// TIA Portal V17 export
// export: Created 2024-09-02T12:50:06.6332122Z, ExportSetting WithDefaults, DisplayName Totally Integrated Automation Portal, DisplayVersion V17, DisplayName TIA Portal Openness, DisplayVersion V17, DisplayName TIA Portal Version Control Interface, DisplayVersion V17, DisplayName STEP 7 Professional, DisplayVersion V17, DisplayName STEP 7 Safety, DisplayVersion V17, DisplayName WinCC Professional, DisplayVersion V17
FUNCTION_BLOCK "GraFB2_FG01_Station_OP70"   // FB1282, GRAPH
VERSION : 0.1
// stored: AcknowledgeErrorsRequired false, AutoNumber false, GraphVersion 4.0, InitialValuesAcquisition true, IsIECCheckEnabled false, LanguageInNetworks LAD, LockOperatingMode false, PermanentILProcessingInMANMode true, SetENOAutomatically false, SkipSteps false, UDAEnableTagReadback false, WithAlarmHandling true
   // inherited from GRAPH_BASE
   VAR
      OFF_SQ_BASE : Bool;
   END_VAR
   VAR_INPUT
      OFF_SQ { ExternalWritable := 'False'} : Bool := false;
      INIT_SQ { ExternalWritable := 'False'} : Bool := false;
      ACK_EF { ExternalWritable := 'False'} : Bool := false;
      S_PREV { ExternalWritable := 'False'} : Bool := false;
      S_NEXT { ExternalWritable := 'False'} : Bool := false;
      SW_AUTO { ExternalWritable := 'False'} : Bool := false;
      SW_TAP { ExternalWritable := 'False'} : Bool := false;
      SW_TOP { ExternalWritable := 'False'} : Bool := false;
      SW_MAN { ExternalWritable := 'False'} : Bool := false;
      S_SEL { ExternalWritable := 'False'} : Int := 0;
      S_ON { ExternalWritable := 'False'} : Bool := false;
      S_OFF { ExternalWritable := 'False'} : Bool := false;
      T_PUSH { ExternalWritable := 'False'} : Bool := false;
   END_VAR
   VAR_OUTPUT
      S_NO { ExternalWritable := 'False'} : Int := 0;
      S_MORE { ExternalWritable := 'False'} : Bool := false;
      S_ACTIVE { ExternalWritable := 'False'} : Bool := false;
      ERR_FLT { ExternalWritable := 'False'} : Bool := false;
      AUTO_ON { ExternalWritable := 'False'} : Bool := false;
      TAP_ON { ExternalWritable := 'False'} : Bool := false;
      TOP_ON { ExternalWritable := 'False'} : Bool := false;
      MAN_ON { ExternalWritable := 'False'} : Bool := false;
   END_VAR
   VAR
      extBlock { S7_SetPoint := 'True'} : "LTLL_ManualGraphExt";
   END_VAR
BEGIN
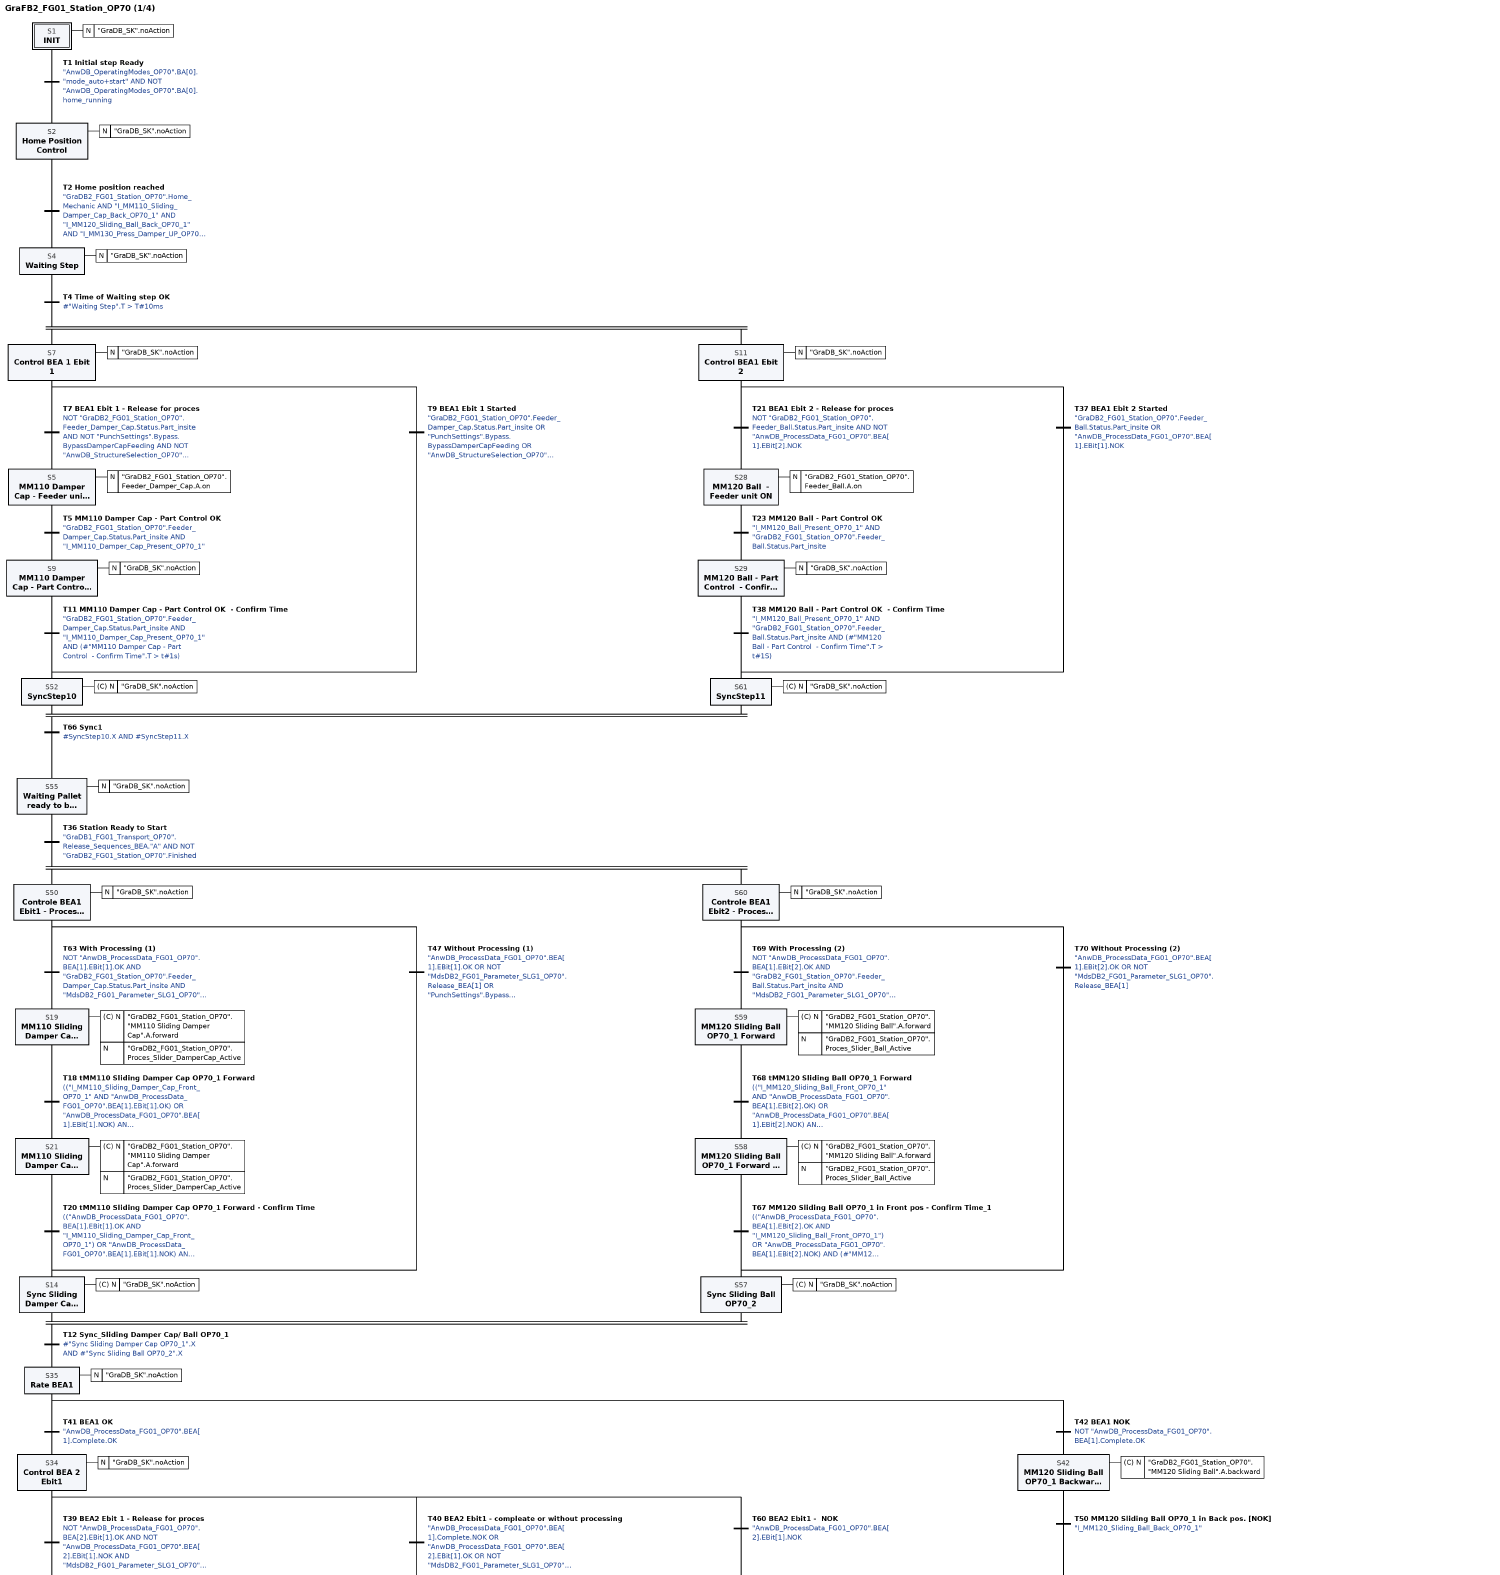
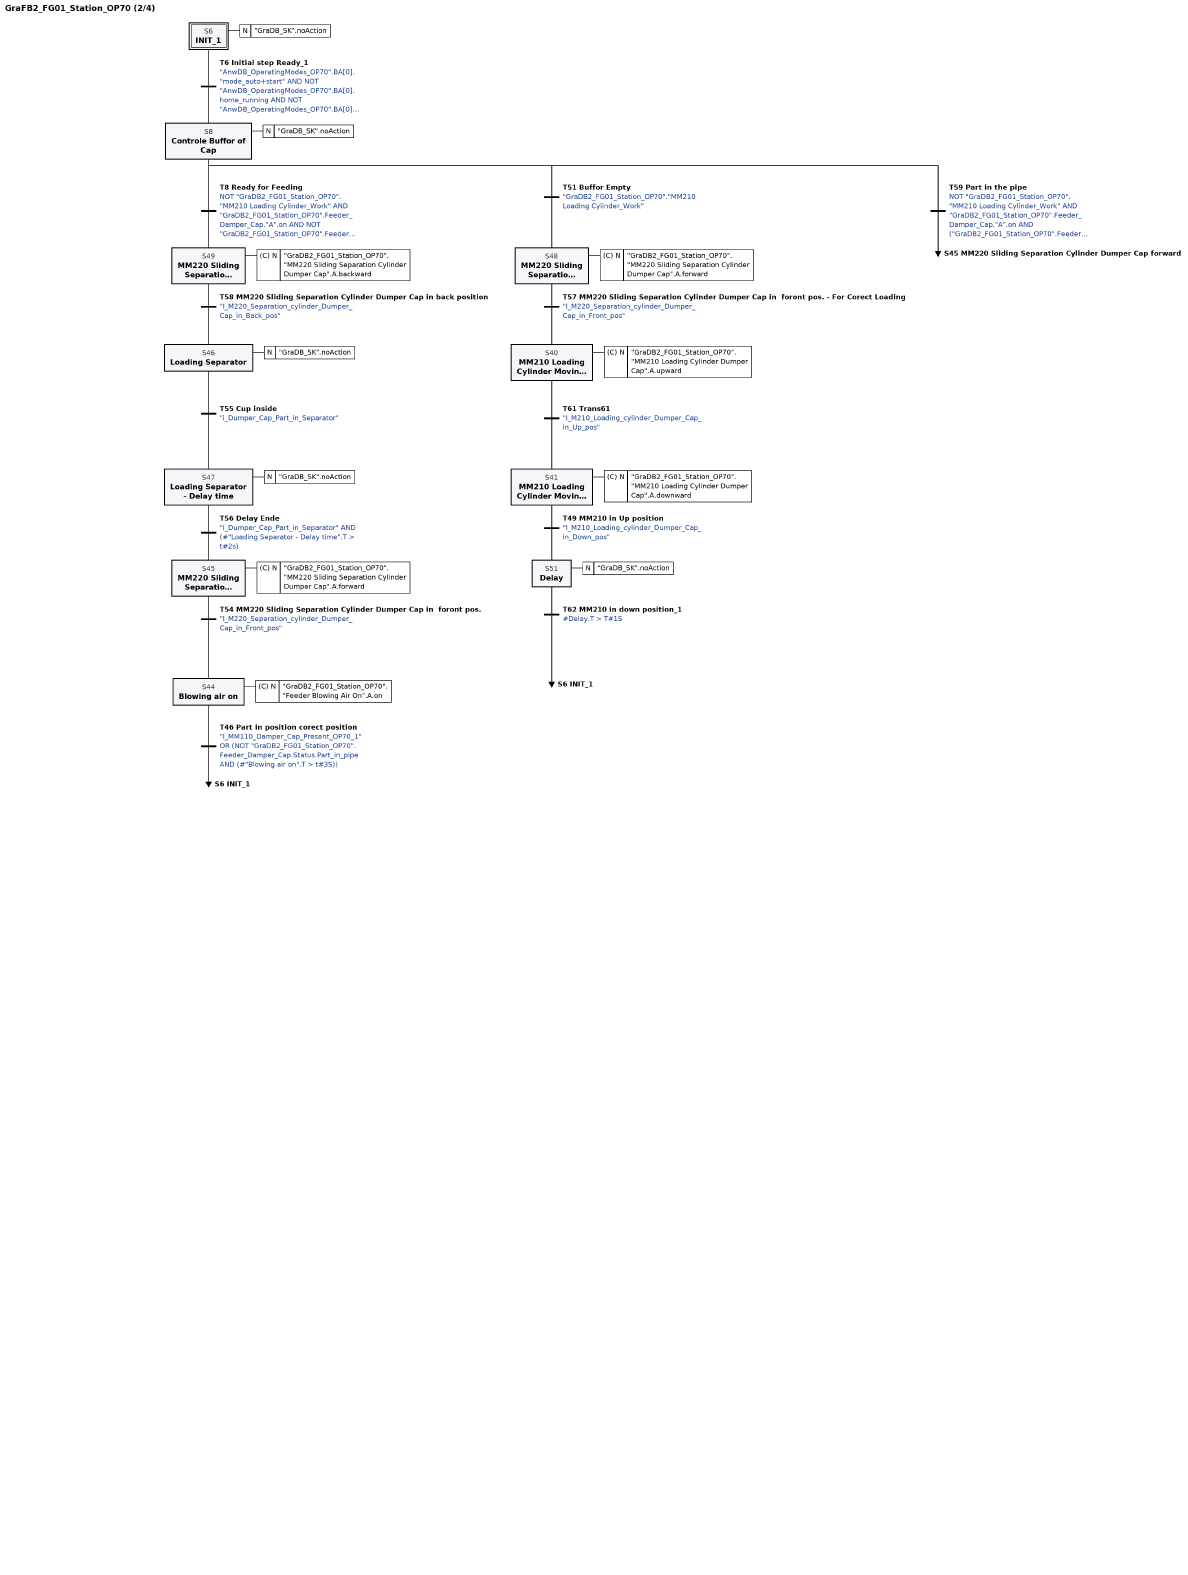
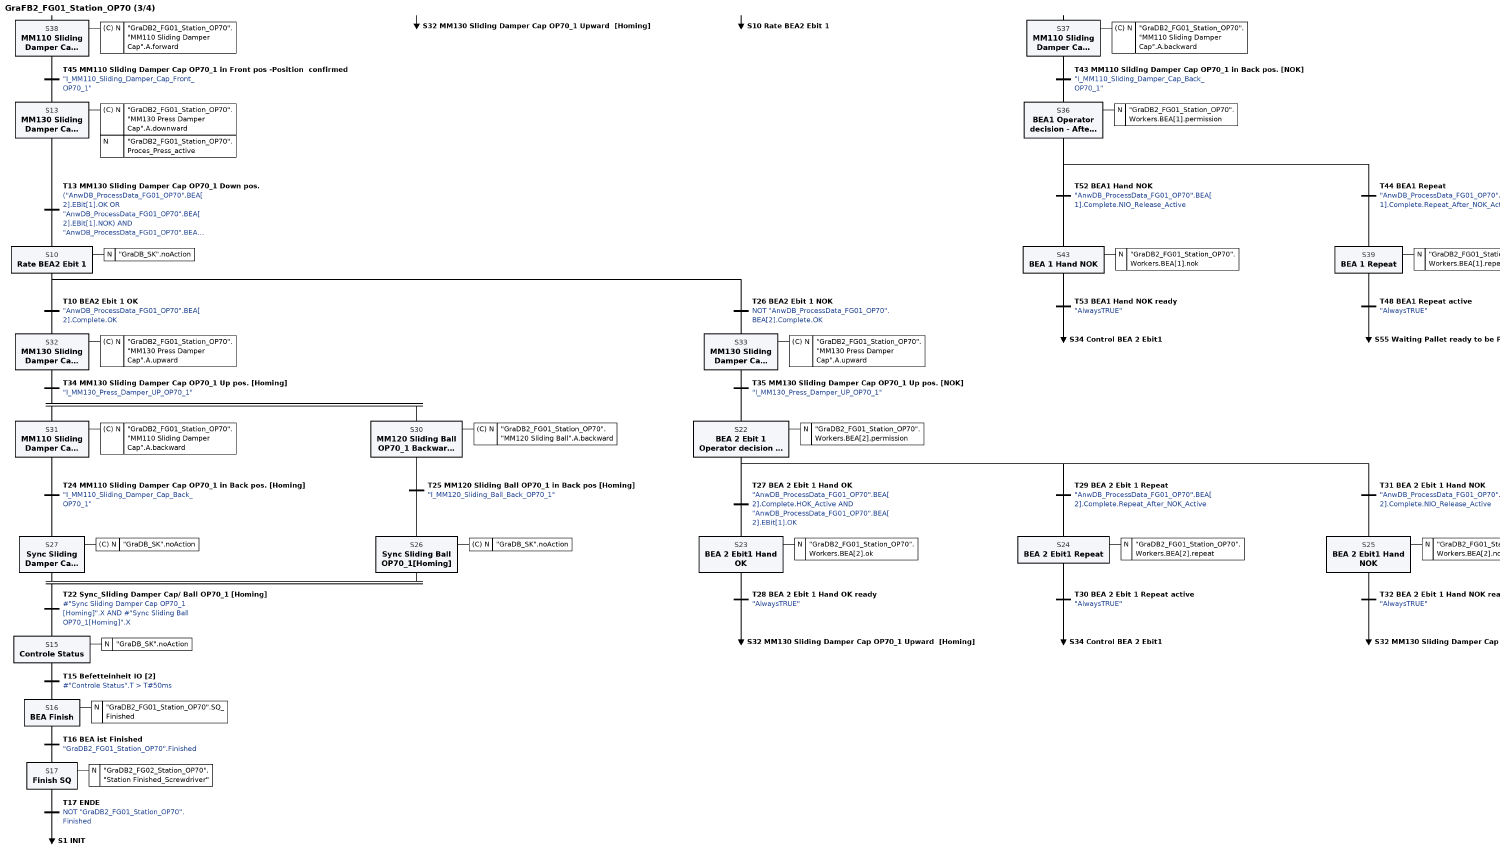
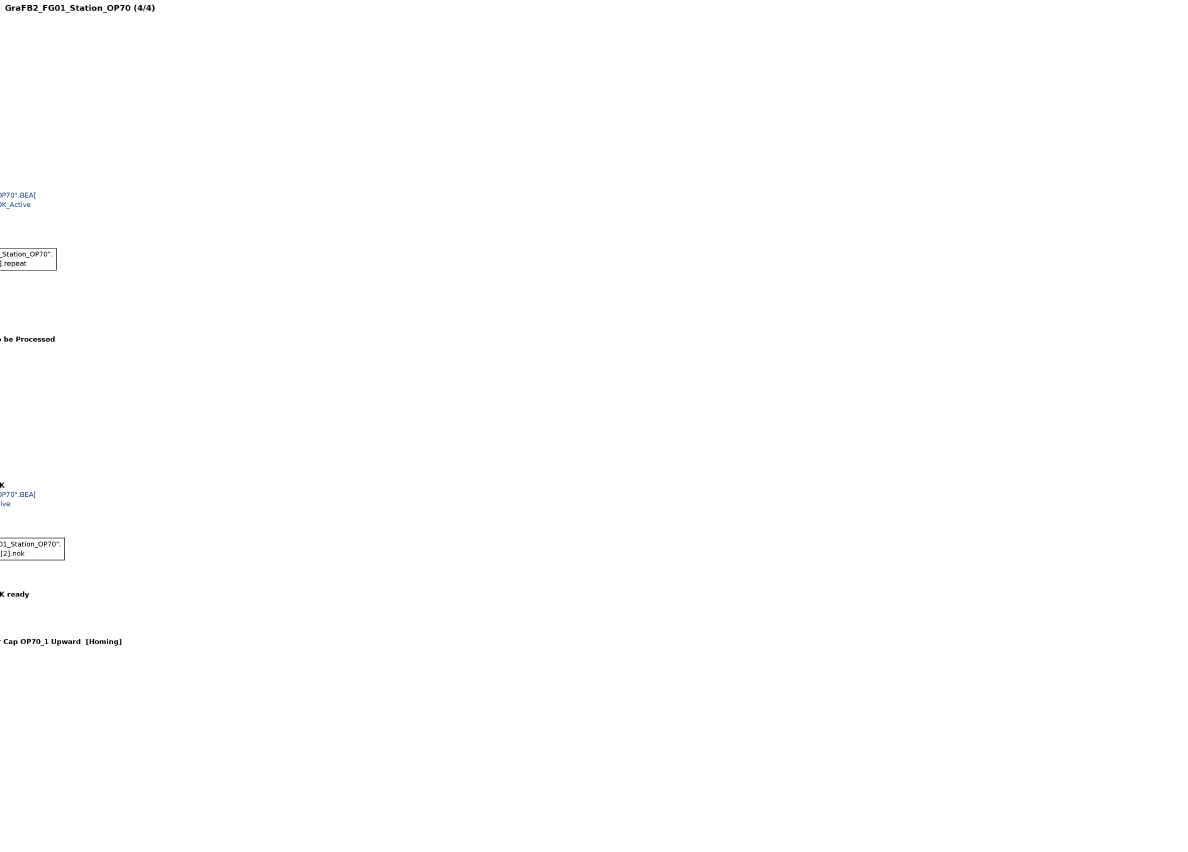
   // permanent pre-instructions
   NETWORK 1
   TITLE = HMI Lite Pass on data
      #extBlock.input := "LTLL_ManualGraphControl_OP70".screen[0].input;
   NETWORK 2
   TITLE = Instance DB Name query and pass on
      GetInstanceName(size := 0, OUT => #extBlock.input.instanceName);
   NETWORK 3
   TITLE = SK Mode
      "SysFC_SQ_Mode"(iFKT := 0, iTmsHalt := false, ioMOP := #RT_DATA.MOP);

   // sequencer 1: Station cycle
   // sample
   INITIAL_STEP INIT:   // S1, max time T#10S, warning time T#7S: Step commentary
      interlock C := (none);   // initial step
      supervision V := (none);   // initial step
              N    "GraDB_SK".noAction
   END_STEP
   TRANSITION "Initial step Ready" FROM INIT TO "Home Position Control"   // T1
      := "AnwDB_OperatingModes_OP70".BA[0]."mode_auto+start" AND NOT "AnwDB_OperatingModes_OP70".BA[0].home_running;
   END_TRANSITION
   STEP "Home Position Control":   // S2, max time T#10S, warning time T#7S
      supervision V := NOT #"Home position reached".TT AND (#"Home Position Control".U > T#1S);
      // Station
              N    "GraDB_SK".noAction
   END_STEP
   TRANSITION "Home position reached" FROM "Home Position Control" TO "Waiting Step"   // T2
      := "GraDB2_FG01_Station_OP70".Home_Mechanic AND "I_MM110_Sliding_Damper_Cap_Back_OP70_1" AND "I_MM120_Sliding_Ball_Back_OP70_1" AND "I_MM130_Press_Damper_UP_OP70_1";
   END_TRANSITION
   STEP "Finish SQ":   // S17, max time T#10S, warning time T#7S
              N    "GraDB2_FG02_Station_OP70"."Station Finished_Screwdriver"
   END_STEP
   TRANSITION ENDE FROM "Finish SQ" TO INIT   // T17, jump
      := NOT "GraDB2_FG01_Station_OP70".Finished;
   END_TRANSITION
   STEP "BEA Finish":   // S16, max time T#10S, warning time T#7S
      supervision V := NOT #"BEA ist Finished".TT AND (#"BEA Finish".U > T#1000ms);
              N    "GraDB2_FG01_Station_OP70".SQ_Finished
   END_STEP
   TRANSITION "BEA ist Finished" FROM "BEA Finish" TO "Finish SQ"   // T16
      := "GraDB2_FG01_Station_OP70".Finished;
   END_TRANSITION
   STEP "Waiting Step":   // S4, max time T#10S, warning time T#7S
      supervision V := NOT #"Time of Waiting step OK".TT AND (#"Waiting Step".U > t#1S);
              N    "GraDB_SK".noAction
   END_STEP
   TRANSITION "Time of Waiting step OK" FROM "Waiting Step" TO ("Control BEA 1 Ebit 1", "Control BEA1 Ebit 2")   // T4
      := #"Waiting Step".T > T#10ms;
   END_TRANSITION
   STEP "Control BEA 1 Ebit 1":   // S7, max time T#10S, warning time T#7S
      supervision V := NOT #"BEA1 Ebit 1 - Release for proces".TT AND (#"Control BEA 1 Ebit 1".U > t#1s);
              N    "GraDB_SK".noAction
   END_STEP
   TRANSITION "BEA1 Ebit 1 - Release for proces" FROM "Control BEA 1 Ebit 1" TO "MM110 Damper Cap - Feeder unit ON"   // T7
      := NOT "GraDB2_FG01_Station_OP70".Feeder_Damper_Cap.Status.Part_insite AND NOT "PunchSettings".Bypass.BypassDamperCapFeeding AND NOT "AnwDB_StructureSelection_OP70".CycleType.Bypass_DamperCaps_FEED AND NOT "AnwDB_ProcessData_FG01_OP70".BEA[1].EBit[1].NOK;
   END_TRANSITION
   TRANSITION "BEA1 Ebit 1 Started" FROM "Control BEA 1 Ebit 1" TO SyncStep10   // T9
      := "GraDB2_FG01_Station_OP70".Feeder_Damper_Cap.Status.Part_insite OR "PunchSettings".Bypass.BypassDamperCapFeeding OR "AnwDB_StructureSelection_OP70".CycleType.Bypass_DamperCaps_FEED OR "AnwDB_ProcessData_FG01_OP70".BEA[1].EBit[1].NOK;
   END_TRANSITION
   STEP "Controle Status":   // S15, max time T#10S, warning time T#7S
      supervision V := NOT #"Befetteinheit IO [2]".TT AND (#"Controle Status".U > T#5s);
              N    "GraDB_SK".noAction
   END_STEP
   TRANSITION "Befetteinheit IO [2]" FROM "Controle Status" TO "BEA Finish"   // T15
      := #"Controle Status".T > T#50ms;
   END_TRANSITION
   STEP "Rate BEA2 Ebit 1":   // S10, max time T#10S, warning time T#7S: When operator access is required
      supervision V := NOT #"BEA2 Ebit 1 OK".TT AND (#"Rate BEA2 Ebit 1".U > t#1s);
              N    "GraDB_SK".noAction
   END_STEP
   TRANSITION "BEA2 Ebit 1 OK" FROM "Rate BEA2 Ebit 1" TO "MM130 Sliding Damper Cap OP70_1 Upward  [Homing]"   // T10
      := "AnwDB_ProcessData_FG01_OP70".BEA[2].Complete.OK;
   END_TRANSITION
   TRANSITION "BEA2 Ebit 1 NOK" FROM "Rate BEA2 Ebit 1" TO "MM130 Sliding Damper Cap OP70_1 Upward  [NOK]"   // T26
      := NOT "AnwDB_ProcessData_FG01_OP70".BEA[2].Complete.OK;
   END_TRANSITION
   STEP "BEA 2 Ebit 1 Operator decision - After NOK":   // S22, max time T#10S, warning time T#7S
      interlock C := "GraDB1_FG01_Transport_OP70".Release_Sequences_BEA."A";
              N    "GraDB2_FG01_Station_OP70".Workers.BEA[2].permission
   END_STEP
   TRANSITION "BEA 2 Ebit 1 Hand OK" FROM "BEA 2 Ebit 1 Operator decision - After NOK" TO "BEA 2 Ebit1 Hand OK"   // T27
      := "AnwDB_ProcessData_FG01_OP70".BEA[2].Complete.HOK_Active AND "AnwDB_ProcessData_FG01_OP70".BEA[2].EBit[1].OK;
   END_TRANSITION
   TRANSITION "BEA 2 Ebit 1 Repeat" FROM "BEA 2 Ebit 1 Operator decision - After NOK" TO "BEA 2 Ebit1 Repeat"   // T29
      := "AnwDB_ProcessData_FG01_OP70".BEA[2].Complete.Repeat_After_NOK_Active;
   END_TRANSITION
   TRANSITION "BEA 2 Ebit 1 Hand NOK" FROM "BEA 2 Ebit 1 Operator decision - After NOK" TO "BEA 2 Ebit1 Hand NOK"   // T31
      := "AnwDB_ProcessData_FG01_OP70".BEA[2].Complete.NIO_Release_Active;
   END_TRANSITION
   STEP "BEA 2 Ebit1 Hand OK":   // S23, max time T#10S, warning time T#7S
              N    "GraDB2_FG01_Station_OP70".Workers.BEA[2].ok
   END_STEP
   TRANSITION "BEA 2 Ebit 1 Hand OK ready" FROM "BEA 2 Ebit1 Hand OK" TO "MM130 Sliding Damper Cap OP70_1 Upward  [Homing]"   // T28, jump
      := "AlwaysTRUE";
   END_TRANSITION
   STEP "BEA 2 Ebit1 Hand NOK":   // S25, max time T#10S, warning time T#7S
              N    "GraDB2_FG01_Station_OP70".Workers.BEA[2].nok
   END_STEP
   TRANSITION "BEA 2 Ebit 1 Hand NOK ready" FROM "BEA 2 Ebit1 Hand NOK" TO "MM130 Sliding Damper Cap OP70_1 Upward  [Homing]"   // T32, jump
      := "AlwaysTRUE";
   END_TRANSITION
   STEP "BEA 2 Ebit1 Repeat":   // S24, max time T#10S, warning time T#7S
              N    "GraDB2_FG01_Station_OP70".Workers.BEA[2].repeat
   END_STEP
   TRANSITION "BEA 2 Ebit 1 Repeat active" FROM "BEA 2 Ebit1 Repeat" TO "Control BEA 2 Ebit1"   // T30, jump
      := "AlwaysTRUE";
   END_TRANSITION
   STEP SyncStep11:   // S61, max time T#10S, warning time T#7S: Step commentary
      interlock C := (none);   // initial step
      supervision V := (none);   // initial step
      (C)     N    "GraDB_SK".noAction
   END_STEP
   STEP "Sync Sliding Damper Cap OP70_1":   // S14, max time T#10S, warning time T#7S: Step commentary
      interlock C := (none);   // initial step
      supervision V := (none);   // initial step
      (C)     N    "GraDB_SK".noAction
   END_STEP
   STEP "MM110 Sliding Damper Cap OP70_1 Forward - Confirm Time":   // S21, max time T#10S, warning time T#7S
      interlock C := "I_MM130_Press_Damper_UP_OP70_1";
      supervision V := NOT #"tMM110 Sliding Damper Cap OP70_1 Forward - Confirm Time".TT AND (#"MM110 Sliding Damper Cap OP70_1 Forward - Confirm Time".U > T#5S);
      (C)     N    "GraDB2_FG01_Station_OP70"."MM110 Sliding Damper Cap".A.forward
              N    "GraDB2_FG01_Station_OP70".Proces_Slider_DamperCap_Active
   END_STEP
   TRANSITION "tMM110 Sliding Damper Cap OP70_1 Forward - Confirm Time" FROM "MM110 Sliding Damper Cap OP70_1 Forward - Confirm Time" TO "Sync Sliding Damper Cap OP70_1"   // T20
      := (("AnwDB_ProcessData_FG01_OP70".BEA[1].EBit[1].OK AND "I_MM110_Sliding_Damper_Cap_Front_OP70_1") OR "AnwDB_ProcessData_FG01_OP70".BEA[1].EBit[1].NOK) AND (#"MM110 Sliding Damper Cap OP70_1 Forward - Confirm Time".T > t#300ms) AND "AnwDB_ProcessData_FG01_OP70".BEA[1].EBit[1].Finished;
   END_TRANSITION
   STEP SyncStep10:   // S52, max time T#10S, warning time T#7S: Step commentary
      interlock C := (none);   // initial step
      supervision V := (none);   // initial step
      (C)     N    "GraDB_SK".noAction
   END_STEP
   TRANSITION Sync1 FROM (SyncStep11, SyncStep10) TO "Waiting Pallet ready to be Processed"   // T66
      := #SyncStep10.X AND #SyncStep11.X;
   END_TRANSITION
   STEP "MM110 Sliding Damper Cap OP70_1 Forward":   // S19, max time T#10S, warning time T#7S
      interlock C := "I_MM130_Press_Damper_UP_OP70_1";
      supervision V := NOT #"tMM110 Sliding Damper Cap OP70_1 Forward".TT AND (#"MM110 Sliding Damper Cap OP70_1 Forward".U > T#5S);
      (C)     N    "GraDB2_FG01_Station_OP70"."MM110 Sliding Damper Cap".A.forward
              N    "GraDB2_FG01_Station_OP70".Proces_Slider_DamperCap_Active
   END_STEP
   TRANSITION "tMM110 Sliding Damper Cap OP70_1 Forward" FROM "MM110 Sliding Damper Cap OP70_1 Forward" TO "MM110 Sliding Damper Cap OP70_1 Forward - Confirm Time"   // T18
      := (("I_MM110_Sliding_Damper_Cap_Front_OP70_1" AND "AnwDB_ProcessData_FG01_OP70".BEA[1].EBit[1].OK) OR "AnwDB_ProcessData_FG01_OP70".BEA[1].EBit[1].NOK) AND "AnwDB_ProcessData_FG01_OP70".BEA[1].EBit[1].Finished;
   END_TRANSITION
   STEP "MM130 Sliding Damper Cap OP70_1 Downward":   // S13, max time T#10S, warning time T#7S
      interlock C := "I_MM110_Sliding_Damper_Cap_Front_OP70_1";
      supervision V := NOT #"MM130 Sliding Damper Cap OP70_1 Down pos.".TT AND (#"MM130 Sliding Damper Cap OP70_1 Downward".U > t#5S);
      (C)     N    "GraDB2_FG01_Station_OP70"."MM130 Press Damper Cap".A.downward
              N    "GraDB2_FG01_Station_OP70".Proces_Press_active
   END_STEP
   TRANSITION "MM130 Sliding Damper Cap OP70_1 Down pos." FROM "MM130 Sliding Damper Cap OP70_1 Downward" TO "Rate BEA2 Ebit 1"   // T13
      := ("AnwDB_ProcessData_FG01_OP70".BEA[2].EBit[1].OK OR "AnwDB_ProcessData_FG01_OP70".BEA[2].EBit[1].NOK) AND "AnwDB_ProcessData_FG01_OP70".BEA[2].EBit[1].Finished;
   END_TRANSITION
   STEP "Sync Sliding Ball OP70_1[Homing]":   // S26, max time T#10S, warning time T#7S: Step commentary
      interlock C := (none);   // initial step
      supervision V := (none);   // initial step
      (C)     N    "GraDB_SK".noAction
   END_STEP
   TRANSITION "Sync_Sliding Damper Cap/ Ball OP70_1 [Homing]" FROM ("Sync Sliding Damper Cap OP70_1 [Homing]", "Sync Sliding Ball OP70_1[Homing]") TO "Controle Status"   // T22
      := #"Sync Sliding Damper Cap OP70_1 [Homing]".X AND #"Sync Sliding Ball OP70_1[Homing]".X;
   END_TRANSITION
   STEP "Sync Sliding Damper Cap OP70_1 [Homing]":   // S27, max time T#10S, warning time T#7S: Step commentary
      interlock C := (none);   // initial step
      supervision V := (none);   // initial step
      (C)     N    "GraDB_SK".noAction
   END_STEP
   STEP "Control BEA 2 Ebit1":   // S34, max time T#10S, warning time T#7S
      supervision V := NOT #"BEA2 Ebit 1 - Release for proces".TT AND (#"Control BEA 2 Ebit1".U > t#1s);
              N    "GraDB_SK".noAction
   END_STEP
   TRANSITION "BEA2 Ebit 1 - Release for proces" FROM "Control BEA 2 Ebit1" TO "MM110 Sliding Damper Cap OP70_1 Forward - Confirm Position before Pressing"   // T39
      := NOT "AnwDB_ProcessData_FG01_OP70".BEA[2].EBit[1].OK AND NOT "AnwDB_ProcessData_FG01_OP70".BEA[2].EBit[1].NOK AND "MdsDB2_FG01_Parameter_SLG1_OP70".Release_BEA[2] AND "AnwDB_ProcessData_FG01_OP70".BEA[1].Complete.OK;
   END_TRANSITION
   TRANSITION "BEA2 Ebit1 - compleate or without processing" FROM "Control BEA 2 Ebit1" TO "MM130 Sliding Damper Cap OP70_1 Upward  [Homing]"   // T40, jump
      := "AnwDB_ProcessData_FG01_OP70".BEA[1].Complete.NOK OR "AnwDB_ProcessData_FG01_OP70".BEA[2].EBit[1].OK OR NOT "MdsDB2_FG01_Parameter_SLG1_OP70".Release_BEA[2];
   END_TRANSITION
   TRANSITION "BEA2 Ebit1 -  NOK" FROM "Control BEA 2 Ebit1" TO "Rate BEA2 Ebit 1"   // T60, jump
      := "AnwDB_ProcessData_FG01_OP70".BEA[2].EBit[1].NOK;
   END_TRANSITION
   STEP "MM110 Damper Cap - Feeder unit ON":   // S5, max time T#10S, warning time T#7S
      supervision V := NOT #"MM110 Damper Cap - Part Control OK".TT AND (#"MM110 Damper Cap - Feeder unit ON".U > t#20S);
              N    "GraDB2_FG01_Station_OP70".Feeder_Damper_Cap.A.on
   END_STEP
   TRANSITION "MM110 Damper Cap - Part Control OK" FROM "MM110 Damper Cap - Feeder unit ON" TO "MM110 Damper Cap - Part Control  - Confirm Time"   // T5
      := "GraDB2_FG01_Station_OP70".Feeder_Damper_Cap.Status.Part_insite AND "I_MM110_Damper_Cap_Present_OP70_1";
   END_TRANSITION
   STEP "MM120 Sliding Ball OP70_1 Backward [Homing]":   // S30, max time T#10S, warning time T#7S
      interlock C := "AlwaysTRUE";
      supervision V := NOT #"MM120 Sliding Ball OP70_1 in Back pos [Homing]".TT AND (#"MM120 Sliding Ball OP70_1 Backward [Homing]".U > T#5S);
      (C)     N    "GraDB2_FG01_Station_OP70"."MM120 Sliding Ball".A.backward
   END_STEP
   TRANSITION "MM120 Sliding Ball OP70_1 in Back pos [Homing]" FROM "MM120 Sliding Ball OP70_1 Backward [Homing]" TO "Sync Sliding Ball OP70_1[Homing]"   // T25
      := "I_MM120_Sliding_Ball_Back_OP70_1";
   END_TRANSITION
   STEP "MM110 Sliding Damper Cap OP70_1 Backward [Homing]":   // S31, max time T#10S, warning time T#7S
      interlock C := "I_MM130_Press_Damper_UP_OP70_1";
      supervision V := NOT #"MM110 Sliding Damper Cap OP70_1 in Back pos. [Homing]".TT AND (#"MM110 Sliding Damper Cap OP70_1 Backward [Homing]".U > T#5S);
      (C)     N    "GraDB2_FG01_Station_OP70"."MM110 Sliding Damper Cap".A.backward
   END_STEP
   TRANSITION "MM110 Sliding Damper Cap OP70_1 in Back pos. [Homing]" FROM "MM110 Sliding Damper Cap OP70_1 Backward [Homing]" TO "Sync Sliding Damper Cap OP70_1 [Homing]"   // T24
      := "I_MM110_Sliding_Damper_Cap_Back_OP70_1";
   END_TRANSITION
   STEP "MM130 Sliding Damper Cap OP70_1 Upward  [Homing]":   // S32, max time T#10S, warning time T#7S
      interlock C := "I_MM110_Sliding_Damper_Cap_Front_OP70_1";
      supervision V := NOT #"MM130 Sliding Damper Cap OP70_1 Up pos. [Homing]".TT AND (#"MM130 Sliding Damper Cap OP70_1 Upward  [Homing]".U > t#1S);
      (C)     N    "GraDB2_FG01_Station_OP70"."MM130 Press Damper Cap".A.upward
   END_STEP
   TRANSITION "MM130 Sliding Damper Cap OP70_1 Up pos. [Homing]" FROM "MM130 Sliding Damper Cap OP70_1 Upward  [Homing]" TO ("MM110 Sliding Damper Cap OP70_1 Backward [Homing]", "MM120 Sliding Ball OP70_1 Backward [Homing]")   // T34
      := "I_MM130_Press_Damper_UP_OP70_1";
   END_TRANSITION
   STEP "MM130 Sliding Damper Cap OP70_1 Upward  [NOK]":   // S33, max time T#10S, warning time T#7S
      interlock C := "I_MM110_Sliding_Damper_Cap_Front_OP70_1";
      supervision V := NOT #"MM130 Sliding Damper Cap OP70_1 Up pos. [NOK]".TT AND (#"MM130 Sliding Damper Cap OP70_1 Upward  [NOK]".U > t#1S);
      (C)     N    "GraDB2_FG01_Station_OP70"."MM130 Press Damper Cap".A.upward
   END_STEP
   TRANSITION "MM130 Sliding Damper Cap OP70_1 Up pos. [NOK]" FROM "MM130 Sliding Damper Cap OP70_1 Upward  [NOK]" TO "BEA 2 Ebit 1 Operator decision - After NOK"   // T35
      := "I_MM130_Press_Damper_UP_OP70_1";
   END_TRANSITION
   STEP "MM110 Damper Cap - Part Control  - Confirm Time":   // S9, max time T#10S, warning time T#7S
      supervision V := NOT #"MM110 Damper Cap - Part Control OK  - Confirm Time".TT AND (#"MM110 Damper Cap - Part Control  - Confirm Time".U > t#1S);
              N    "GraDB_SK".noAction
   END_STEP
   TRANSITION "MM110 Damper Cap - Part Control OK  - Confirm Time" FROM "MM110 Damper Cap - Part Control  - Confirm Time" TO SyncStep10   // T11
      := "GraDB2_FG01_Station_OP70".Feeder_Damper_Cap.Status.Part_insite AND "I_MM110_Damper_Cap_Present_OP70_1" AND (#"MM110 Damper Cap - Part Control  - Confirm Time".T > t#1s);
   END_TRANSITION
   STEP "Control BEA1 Ebit 2":   // S11, max time T#10S, warning time T#7S
      supervision V := NOT #"BEA1 Ebit 2 - Release for proces".TT AND (#"Control BEA1 Ebit 2".U > t#1s);
              N    "GraDB_SK".noAction
   END_STEP
   TRANSITION "BEA1 Ebit 2 - Release for proces" FROM "Control BEA1 Ebit 2" TO "MM120 Ball  - Feeder unit ON"   // T21
      := NOT "GraDB2_FG01_Station_OP70".Feeder_Ball.Status.Part_insite AND NOT "AnwDB_ProcessData_FG01_OP70".BEA[1].EBit[2].NOK;
   END_TRANSITION
   TRANSITION "BEA1 Ebit 2 Started" FROM "Control BEA1 Ebit 2" TO SyncStep11   // T37
      := "GraDB2_FG01_Station_OP70".Feeder_Ball.Status.Part_insite OR "AnwDB_ProcessData_FG01_OP70".BEA[1].EBit[1].NOK;
   END_TRANSITION
   STEP "MM120 Ball  - Feeder unit ON":   // S28, max time T#10S, warning time T#7S
      supervision V := NOT #"MM120 Ball - Part Control OK".TT AND (#"MM120 Ball  - Feeder unit ON".U > t#7s);
              N    "GraDB2_FG01_Station_OP70".Feeder_Ball.A.on
   END_STEP
   TRANSITION "MM120 Ball - Part Control OK" FROM "MM120 Ball  - Feeder unit ON" TO "MM120 Ball - Part Control  - Confirm Time"   // T23
      := "I_MM120_Ball_Present_OP70_1" AND "GraDB2_FG01_Station_OP70".Feeder_Ball.Status.Part_insite;
   END_TRANSITION
   STEP "MM120 Ball - Part Control  - Confirm Time":   // S29, max time T#10S, warning time T#7S
      supervision V := NOT #"MM120 Ball - Part Control OK  - Confirm Time".TT AND (#"MM120 Ball - Part Control  - Confirm Time".U > t#1S);
              N    "GraDB_SK".noAction
   END_STEP
   TRANSITION "MM120 Ball - Part Control OK  - Confirm Time" FROM "MM120 Ball - Part Control  - Confirm Time" TO SyncStep11   // T38
      := "I_MM120_Ball_Present_OP70_1" AND "GraDB2_FG01_Station_OP70".Feeder_Ball.Status.Part_insite AND (#"MM120 Ball - Part Control  - Confirm Time".T > t#1S);
   END_TRANSITION
   STEP "MM120 Sliding Ball OP70_1 Backward [NOK]":   // S42, max time T#10S, warning time T#7S
      interlock C := "I_MM130_Press_Damper_UP_OP70_1";
      supervision V := NOT #"MM120 Sliding Ball OP70_1 in Back pos. [NOK]".TT AND (#"MM120 Sliding Ball OP70_1 Backward [NOK]".U > T#5S);
      (C)     N    "GraDB2_FG01_Station_OP70"."MM120 Sliding Ball".A.backward
   END_STEP
   TRANSITION "MM120 Sliding Ball OP70_1 in Back pos. [NOK]" FROM "MM120 Sliding Ball OP70_1 Backward [NOK]" TO "MM110 Sliding Damper Cap OP70_1 Backward [NOK]"   // T50
      := "I_MM120_Sliding_Ball_Back_OP70_1";
   END_TRANSITION
   STEP "Rate BEA1":   // S35, max time T#10S, warning time T#7S: When operator access is required
      supervision V := NOT #"BEA1 OK".TT AND (#"Rate BEA1".U > t#1s);
              N    "GraDB_SK".noAction
   END_STEP
   TRANSITION "BEA1 OK" FROM "Rate BEA1" TO "Control BEA 2 Ebit1"   // T41
      := "AnwDB_ProcessData_FG01_OP70".BEA[1].Complete.OK;
   END_TRANSITION
   TRANSITION "BEA1 NOK" FROM "Rate BEA1" TO "MM120 Sliding Ball OP70_1 Backward [NOK]"   // T42
      := NOT "AnwDB_ProcessData_FG01_OP70".BEA[1].Complete.OK;
   END_TRANSITION
   STEP "BEA1 Operator decision - After NOK":   // S36, max time T#10S, warning time T#7S
      interlock C := "GraDB1_FG01_Transport_OP70".Release_Sequences_BEA."A";
              N    "GraDB2_FG01_Station_OP70".Workers.BEA[1].permission
   END_STEP
   TRANSITION "BEA1 Hand NOK" FROM "BEA1 Operator decision - After NOK" TO "BEA 1 Hand NOK"   // T52
      := "AnwDB_ProcessData_FG01_OP70".BEA[1].Complete.NIO_Release_Active;
   END_TRANSITION
   TRANSITION "BEA1 Repeat" FROM "BEA1 Operator decision - After NOK" TO "BEA 1 Repeat"   // T44
      := "AnwDB_ProcessData_FG01_OP70".BEA[1].Complete.Repeat_After_NOK_Active;
   END_TRANSITION
   STEP "MM110 Sliding Damper Cap OP70_1 Backward [NOK]":   // S37, max time T#10S, warning time T#7S
      interlock C := "I_MM130_Press_Damper_UP_OP70_1";
      supervision V := NOT #"MM110 Sliding Damper Cap OP70_1 in Back pos. [NOK]".TT AND (#"MM110 Sliding Damper Cap OP70_1 Backward [NOK]".U > T#5S);
      (C)     N    "GraDB2_FG01_Station_OP70"."MM110 Sliding Damper Cap".A.backward
   END_STEP
   TRANSITION "MM110 Sliding Damper Cap OP70_1 in Back pos. [NOK]" FROM "MM110 Sliding Damper Cap OP70_1 Backward [NOK]" TO "BEA1 Operator decision - After NOK"   // T43
      := "I_MM110_Sliding_Damper_Cap_Back_OP70_1";
   END_TRANSITION
   STEP "BEA 1 Repeat":   // S39, max time T#10S, warning time T#7S
              N    "GraDB2_FG01_Station_OP70".Workers.BEA[1].repeat
   END_STEP
   TRANSITION "BEA1 Repeat active" FROM "BEA 1 Repeat" TO "Waiting Pallet ready to be Processed"   // T48, jump
      := "AlwaysTRUE";
   END_TRANSITION
   STEP "BEA 1 Hand NOK":   // S43, max time T#10S, warning time T#7S
              N    "GraDB2_FG01_Station_OP70".Workers.BEA[1].nok
   END_STEP
   TRANSITION "BEA1 Hand NOK ready" FROM "BEA 1 Hand NOK" TO "Control BEA 2 Ebit1"   // T53, jump
      := "AlwaysTRUE";
   END_TRANSITION
   STEP "MM110 Sliding Damper Cap OP70_1 Forward - Confirm Position before Pressing":   // S38, max time T#10S, warning time T#7S
      interlock C := "I_MM130_Press_Damper_UP_OP70_1";
      supervision V := NOT #"MM110 Sliding Damper Cap OP70_1 in Front pos -Position  confirmed".TT AND (#"MM110 Sliding Damper Cap OP70_1 Forward - Confirm Position before Pressing".U > T#5S);
      (C)     N    "GraDB2_FG01_Station_OP70"."MM110 Sliding Damper Cap".A.forward
   END_STEP
   TRANSITION "MM110 Sliding Damper Cap OP70_1 in Front pos -Position  confirmed" FROM "MM110 Sliding Damper Cap OP70_1 Forward - Confirm Position before Pressing" TO "MM130 Sliding Damper Cap OP70_1 Downward"   // T45
      := "I_MM110_Sliding_Damper_Cap_Front_OP70_1";
   END_TRANSITION
   STEP "Controle BEA1 Ebit1 - Process Release":   // S50, max time T#10S, warning time T#7S
      supervision V := NOT #"BEA1 Ebit 1 - Release for proces".TT AND (#"Controle BEA1 Ebit1 - Process Release".U > t#1s);
              N    "GraDB_SK".noAction
   END_STEP
   TRANSITION "With Processing (1)" FROM "Controle BEA1 Ebit1 - Process Release" TO "MM110 Sliding Damper Cap OP70_1 Forward"   // T63
      := NOT "AnwDB_ProcessData_FG01_OP70".BEA[1].EBit[1].OK AND "GraDB2_FG01_Station_OP70".Feeder_Damper_Cap.Status.Part_insite AND "MdsDB2_FG01_Parameter_SLG1_OP70".Release_BEA[1] AND NOT "PunchSettings".Bypass.BypassDamperCapFeeding AND NOT "AnwDB_StructureSelection_OP70".CycleType.Bypass_DamperCaps_FEED;
   END_TRANSITION
   TRANSITION "Without Processing (1)" FROM "Controle BEA1 Ebit1 - Process Release" TO "Sync Sliding Damper Cap OP70_1"   // T47
      := "AnwDB_ProcessData_FG01_OP70".BEA[1].EBit[1].OK OR NOT "MdsDB2_FG01_Parameter_SLG1_OP70".Release_BEA[1] OR "PunchSettings".Bypass.BypassDamperCapFeeding OR "AnwDB_StructureSelection_OP70".CycleType.Bypass_DamperCaps_FEED;
   END_TRANSITION
   STEP "Waiting Pallet ready to be Processed":   // S55, max time T#10S, warning time T#7S
              N    "GraDB_SK".noAction
   END_STEP
   TRANSITION "Station Ready to Start" FROM "Waiting Pallet ready to be Processed" TO ("Controle BEA1 Ebit1 - Process Release", "Controle BEA1 Ebit2 - Process Release")   // T36
      := "GraDB1_FG01_Transport_OP70".Release_Sequences_BEA."A" AND NOT "GraDB2_FG01_Station_OP70".Finished;
   END_TRANSITION
   STEP "Sync Sliding Ball OP70_2":   // S57, max time T#10S, warning time T#7S: Step commentary
      interlock C := (none);   // initial step
      supervision V := (none);   // initial step
      (C)     N    "GraDB_SK".noAction
   END_STEP
   TRANSITION "Sync_Sliding Damper Cap/ Ball OP70_1" FROM ("Sync Sliding Damper Cap OP70_1", "Sync Sliding Ball OP70_2") TO "Rate BEA1"   // T12
      := #"Sync Sliding Damper Cap OP70_1".X AND #"Sync Sliding Ball OP70_2".X;
   END_TRANSITION
   STEP "MM120 Sliding Ball OP70_1 Forward - Confirm Time":   // S58, max time T#10S, warning time T#7S
      interlock C := "AlwaysTRUE";
      supervision V := NOT #"MM120 Sliding Ball OP70_1 in Front pos - Confirm Time_1".TT AND (#"MM120 Sliding Ball OP70_1 Forward - Confirm Time".U > T#5S);
      (C)     N    "GraDB2_FG01_Station_OP70"."MM120 Sliding Ball".A.forward
              N    "GraDB2_FG01_Station_OP70".Proces_Slider_Ball_Active
   END_STEP
   TRANSITION "MM120 Sliding Ball OP70_1 in Front pos - Confirm Time_1" FROM "MM120 Sliding Ball OP70_1 Forward - Confirm Time" TO "Sync Sliding Ball OP70_2"   // T67
      := (("AnwDB_ProcessData_FG01_OP70".BEA[1].EBit[2].OK AND "I_MM120_Sliding_Ball_Front_OP70_1") OR "AnwDB_ProcessData_FG01_OP70".BEA[1].EBit[2].NOK) AND (#"MM120 Sliding Ball OP70_1 Forward - Confirm Time".T > t#300ms) AND "AnwDB_ProcessData_FG01_OP70".BEA[1].EBit[2].Finished;
   END_TRANSITION
   STEP "MM120 Sliding Ball OP70_1 Forward":   // S59, max time T#10S, warning time T#7S
      interlock C := "AlwaysTRUE";
      supervision V := NOT #"tMM120 Sliding Ball OP70_1 Forward".TT AND (#"MM120 Sliding Ball OP70_1 Forward".U > T#5S);
      (C)     N    "GraDB2_FG01_Station_OP70"."MM120 Sliding Ball".A.forward
              N    "GraDB2_FG01_Station_OP70".Proces_Slider_Ball_Active
   END_STEP
   TRANSITION "tMM120 Sliding Ball OP70_1 Forward" FROM "MM120 Sliding Ball OP70_1 Forward" TO "MM120 Sliding Ball OP70_1 Forward - Confirm Time"   // T68
      := (("I_MM120_Sliding_Ball_Front_OP70_1" AND "AnwDB_ProcessData_FG01_OP70".BEA[1].EBit[2].OK) OR "AnwDB_ProcessData_FG01_OP70".BEA[1].EBit[2].NOK) AND "AnwDB_ProcessData_FG01_OP70".BEA[1].EBit[2].Finished;
   END_TRANSITION
   STEP "Controle BEA1 Ebit2 - Process Release":   // S60, max time T#10S, warning time T#7S
      supervision V := NOT #"BEA1 Ebit 1 - Release for proces".TT AND (#"Controle BEA1 Ebit2 - Process Release".U > t#1s);
              N    "GraDB_SK".noAction
   END_STEP
   TRANSITION "With Processing (2)" FROM "Controle BEA1 Ebit2 - Process Release" TO "MM120 Sliding Ball OP70_1 Forward"   // T69
      := NOT "AnwDB_ProcessData_FG01_OP70".BEA[1].EBit[2].OK AND "GraDB2_FG01_Station_OP70".Feeder_Ball.Status.Part_insite AND "MdsDB2_FG01_Parameter_SLG1_OP70".Release_BEA[1];
   END_TRANSITION
   TRANSITION "Without Processing (2)" FROM "Controle BEA1 Ebit2 - Process Release" TO "Sync Sliding Ball OP70_2"   // T70
      := "AnwDB_ProcessData_FG01_OP70".BEA[1].EBit[2].OK OR NOT "MdsDB2_FG01_Parameter_SLG1_OP70".Release_BEA[1];
   END_TRANSITION

   // sequencer 2: FeederUnit
   STEP "Controle Buffor of Cap":   // S8, max time T#10S, warning time T#7S
              N    "GraDB_SK".noAction
   END_STEP
   TRANSITION "Ready for Feeding" FROM "Controle Buffor of Cap" TO "MM220 Sliding Separation Cylinder Dumper Cap Backward - for picking"   // T8
      := NOT "GraDB2_FG01_Station_OP70"."MM210 Loading Cylinder_Work" AND "GraDB2_FG01_Station_OP70".Feeder_Damper_Cap."A".on AND NOT "GraDB2_FG01_Station_OP70".Feeder_Damper_Cap.Status.Part_in_Separator AND NOT "GraDB2_FG01_Station_OP70".Feeder_Damper_Cap.Status.Part_in_pipe AND NOT "GraDB2_FG01_Station_OP70".Feeder_Damper_Cap.Status.Part_insite AND NOT "AnwDB_ProcessData_FG01_OP70".BEA[1].EBit[1].NOK;
   END_TRANSITION
   TRANSITION "Buffor Empty" FROM "Controle Buffor of Cap" TO "MM220 Sliding Separation Cylinder Dumper Cap forward - For Corect Loading"   // T51
      := "GraDB2_FG01_Station_OP70"."MM210 Loading Cylinder_Work";
   END_TRANSITION
   TRANSITION "Part in the pipe" FROM "Controle Buffor of Cap" TO "MM220 Sliding Separation Cylinder Dumper Cap forward"   // T59, jump
      := NOT "GraDB2_FG01_Station_OP70"."MM210 Loading Cylinder_Work" AND "GraDB2_FG01_Station_OP70".Feeder_Damper_Cap."A".on AND ("GraDB2_FG01_Station_OP70".Feeder_Damper_Cap.Status.Part_in_Separator OR "GraDB2_FG01_Station_OP70".Feeder_Damper_Cap.Status.Part_in_pipe) AND NOT "GraDB2_FG01_Station_OP70".Feeder_Damper_Cap.Status.Part_insite AND NOT "AnwDB_ProcessData_FG01_OP70".BEA[1].EBit[1].NOK;
   END_TRANSITION
   INITIAL_STEP INIT_1:   // S6, max time T#10S, warning time T#7S: Step commentary
      interlock C := (none);   // initial step
      supervision V := (none);   // initial step
              N    "GraDB_SK".noAction
   END_STEP
   TRANSITION "Initial step Ready_1" FROM INIT_1 TO "Controle Buffor of Cap"   // T6
      := "AnwDB_OperatingModes_OP70".BA[0]."mode_auto+start" AND NOT "AnwDB_OperatingModes_OP70".BA[0].home_running AND NOT "AnwDB_OperatingModes_OP70".BA[0].tacte_end;
   END_TRANSITION
   STEP "MM210 Loading Cylinder Moving Upward_":   // S40, max time T#10S, warning time T#7S
      (C)     N    "GraDB2_FG01_Station_OP70"."MM210 Loading Cylinder Dumper Cap".A.upward
   END_STEP
   TRANSITION Trans61 FROM "MM210 Loading Cylinder Moving Upward_" TO "MM210 Loading Cylinder Moving Downward"   // T61
      := "I_M210_Loading_cylinder_Dumper_Cap_in_Up_pos";
   END_TRANSITION
   STEP "MM210 Loading Cylinder Moving Downward":   // S41, max time T#10S, warning time T#7S
      (C)     N    "GraDB2_FG01_Station_OP70"."MM210 Loading Cylinder Dumper Cap".A.downward
   END_STEP
   TRANSITION "MM210 in Up position" FROM "MM210 Loading Cylinder Moving Downward" TO Delay   // T49
      := "I_M210_Loading_cylinder_Dumper_Cap_in_Down_pos";
   END_TRANSITION
   STEP "Blowing air on":   // S44, max time T#10S, warning time T#7S
      supervision V := NOT #"Part in position corect position".TT AND (#"Blowing air on".U > T#5S);
      (C)     N    "GraDB2_FG01_Station_OP70"."Feeder Blowing Air On".A.on
   END_STEP
   TRANSITION "Part in position corect position" FROM "Blowing air on" TO INIT_1   // T46, jump
      := "I_MM110_Damper_Cap_Present_OP70_1" OR (NOT "GraDB2_FG01_Station_OP70".Feeder_Damper_Cap.Status.Part_in_pipe AND (#"Blowing air on".T > t#3S));
   END_TRANSITION
   STEP "MM220 Sliding Separation Cylinder Dumper Cap forward":   // S45, max time T#10S, warning time T#7S
      supervision V := NOT #"MM220 Sliding Separation Cylinder Dumper Cap in  foront pos.".TT AND (#"MM220 Sliding Separation Cylinder Dumper Cap forward".U > t#2S);
      (C)     N    "GraDB2_FG01_Station_OP70"."MM220 Sliding Separation Cylinder Dumper Cap".A.forward
   END_STEP
   TRANSITION "MM220 Sliding Separation Cylinder Dumper Cap in  foront pos." FROM "MM220 Sliding Separation Cylinder Dumper Cap forward" TO "Blowing air on"   // T54
      := "I_M220_Separation_cylinder_Dumper_Cap_in_Front_pos";
   END_TRANSITION
   STEP "Loading Separator":   // S46, max time T#10S, warning time T#7S
              N    "GraDB_SK".noAction
   END_STEP
   TRANSITION "Cup inside" FROM "Loading Separator" TO "Loading Separator - Delay time"   // T55
      := "i_Dumper_Cap_Part_in_Separator";
   END_TRANSITION
   STEP "Loading Separator - Delay time":   // S47, max time T#10S, warning time T#7S
              N    "GraDB_SK".noAction
   END_STEP
   TRANSITION "Delay Ende" FROM "Loading Separator - Delay time" TO "MM220 Sliding Separation Cylinder Dumper Cap forward"   // T56
      := "i_Dumper_Cap_Part_in_Separator" AND (#"Loading Separator - Delay time".T > t#2s);
   END_TRANSITION
   STEP "MM220 Sliding Separation Cylinder Dumper Cap Backward - for picking":   // S49, max time T#10S, warning time T#7S
      interlock C := NOT "GraDB2_FG01_Station_OP70".Feeder_Damper_Cap.Status.Part_in_Separator AND NOT "GraDB2_FG01_Station_OP70".Feeder_Damper_Cap.Status.Part_in_pipe;
      supervision V := NOT #"MM220 Sliding Separation Cylinder Dumper Cap in back position".TT AND (#"MM220 Sliding Separation Cylinder Dumper Cap Backward - for picking".U > t#2S);
      (C)     N    "GraDB2_FG01_Station_OP70"."MM220 Sliding Separation Cylinder Dumper Cap".A.backward
   END_STEP
   TRANSITION "MM220 Sliding Separation Cylinder Dumper Cap in back position" FROM "MM220 Sliding Separation Cylinder Dumper Cap Backward - for picking" TO "Loading Separator"   // T58
      := "I_M220_Separation_cylinder_Dumper_Cap_in_Back_pos";
   END_TRANSITION
   STEP "MM220 Sliding Separation Cylinder Dumper Cap forward - For Corect Loading":   // S48, max time T#10S, warning time T#7S
      supervision V := NOT #"MM220 Sliding Separation Cylinder Dumper Cap in  foront pos. - For Corect Loading".TT AND (#"MM220 Sliding Separation Cylinder Dumper Cap forward - For Corect Loading".U > t#2S);
      (C)     N    "GraDB2_FG01_Station_OP70"."MM220 Sliding Separation Cylinder Dumper Cap".A.forward
   END_STEP
   TRANSITION "MM220 Sliding Separation Cylinder Dumper Cap in  foront pos. - For Corect Loading" FROM "MM220 Sliding Separation Cylinder Dumper Cap forward - For Corect Loading" TO "MM210 Loading Cylinder Moving Upward_"   // T57
      := "I_M220_Separation_cylinder_Dumper_Cap_in_Front_pos";
   END_TRANSITION
   STEP Delay:   // S51, max time T#10S, warning time T#7S
              N    "GraDB_SK".noAction
   END_STEP
   TRANSITION "MM210 in down position_1" FROM Delay TO INIT_1   // T62, jump
      := #Delay.T > T#1S;
   END_TRANSITION

   // permanent post-instructions
   NETWORK 1
   TITLE = Move interlocks from Ext block to ManualGraphControl DB
      "LTLL_ManualGraphInterlock"(ManualGraphExtOutput := #extBlock.output,
                              ManualGraphControlScreen := "LTLL_ManualGraphControl_OP70".screen[0]);
   NETWORK 2
   TITLE = Report step error
      "SysFC_NumOfSQErrors"(FLT := #RT_DATA.SQ_FLAGS.ERR_FLT,
                            Fault_SQ := "AnwDB_OperatingModes_OP70".BA[0].error_report_SK,
                            NumOf_Fault_SQ := "AnwDB_ZP_Alarm_OP70".FaultsNoSK_ST1);
   NETWORK 3
   TITLE = Basic position Step chain
      "GraDB2_FG01_Station_OP70".Home_SQ := #INIT.X OR #"Waiting Pallet ready to be Processed".X OR #"Finish SQ".X OR #"Waiting Pallet ready to be Processed".X;
END_FUNCTION_BLOCK
